# EPICS substitutions: src/makeBaseApp/top/pcdsIocApp/archiveSrc/archive__APPNAME_.substitutions
#
# _APPNAME_ substitutions file
#

# Generate iocAdmin archive request
file archive_iocAdmin.template
{
	{
		# Hack till msi supports empty substitutions
		_FOOBAR_=_FOOBAR_
	}
}
